// TIA Portal V19 export
FUNCTION "FC_EM_Plate" : Void   // FC4, FBD
{ S7_Optimized_Access := 'TRUE' }
// stored: SetENOAutomatically false
   VAR_TEMP
      Debug : Bool;
   END_VAR
BEGIN

REGION Network 1: ------------------------------------------------------------------------ Inputs ------------------------------------------------------------------------
END_REGION

REGION Network 2: Verwerken iPlateSenCilPushingIn_d0
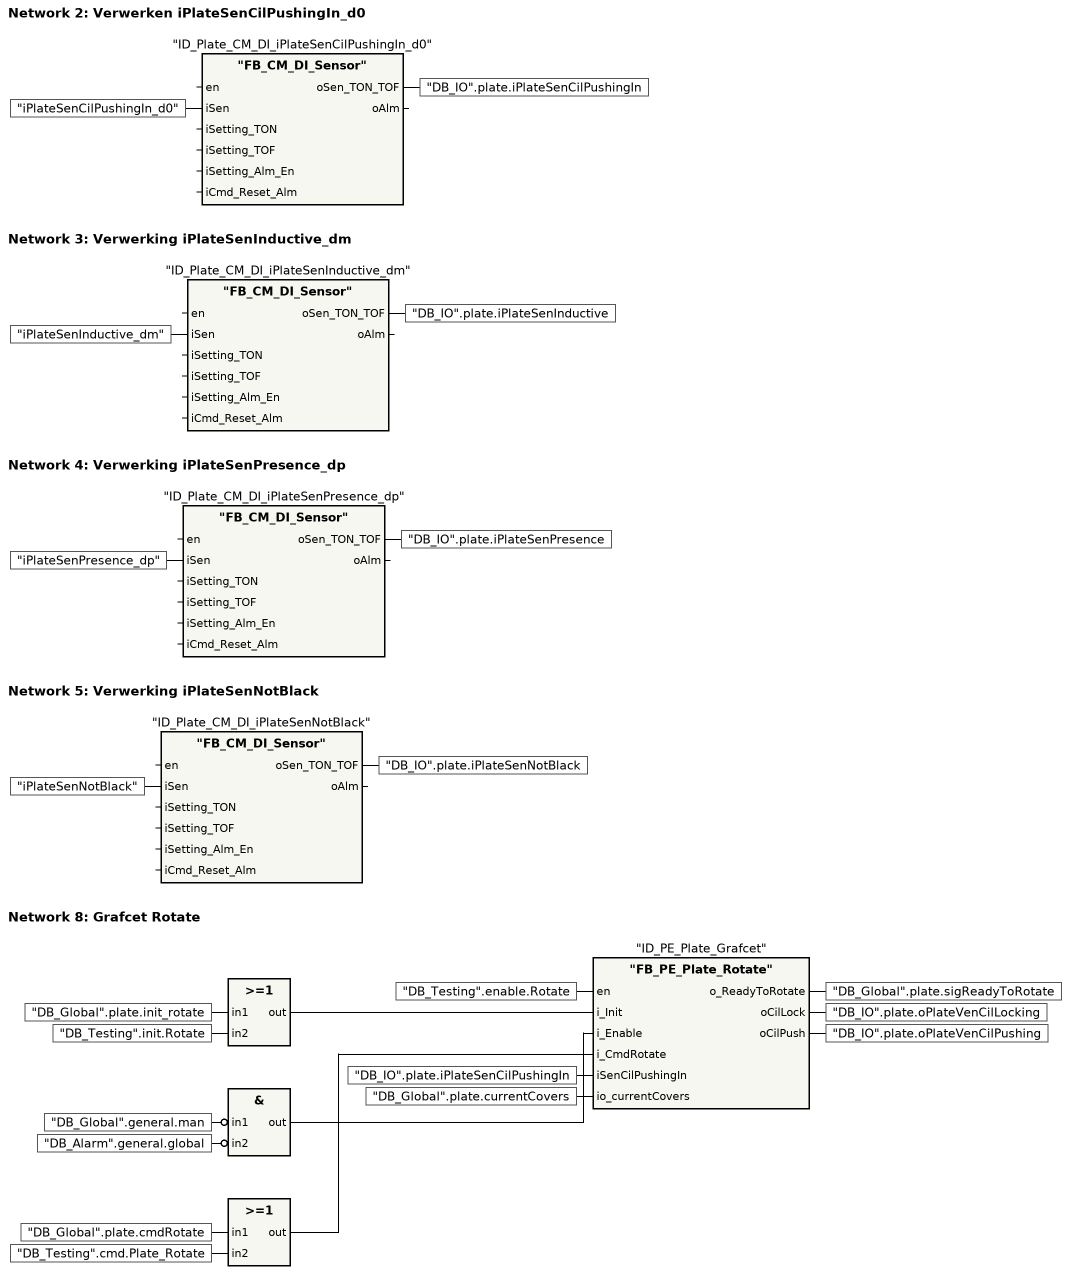
   "ID_Plate_CM_DI_iPlateSenCilPushingIn_d0"(iSen := "iPlateSenCilPushingIn_d0",   // "FB_CM_DI_Sensor"
                           oSen_TON_TOF => "DB_IO".plate.iPlateSenCilPushingIn);
END_REGION

REGION Network 3: Verwerking iPlateSenInductive_dm
   "ID_Plate_CM_DI_iPlateSenInductive_dm"(iSen := "iPlateSenInductive_dm",   // "FB_CM_DI_Sensor"
                           oSen_TON_TOF => "DB_IO".plate.iPlateSenInductive);
END_REGION

REGION Network 4: Verwerking iPlateSenPresence_dp
   "ID_Plate_CM_DI_iPlateSenPresence_dp"(iSen := "iPlateSenPresence_dp",   // "FB_CM_DI_Sensor"
                           oSen_TON_TOF => "DB_IO".plate.iPlateSenPresence);
END_REGION

REGION Network 5: Verwerking iPlateSenNotBlack
   "ID_Plate_CM_DI_iPlateSenNotBlack"(iSen := "iPlateSenNotBlack",   // "FB_CM_DI_Sensor"
                           oSen_TON_TOF => "DB_IO".plate.iPlateSenNotBlack);
END_REGION

REGION Network 6 (SCL): Verwerking iPlateSenHeight
   "DB_IO".plate.iPlateSenHeight := "iPlateSenHeight";
END_REGION

REGION Network 7: ------------------------------------------------------------------------ Logic ------------------------------------------------------------------------
END_REGION

REGION Network 8: Grafcet Rotate
   IF "DB_Testing".enable.Rotate THEN
       "ID_PE_Plate_Grafcet"(i_Init := "DB_Global".plate.init_rotate OR "DB_Testing".init.Rotate,   // "FB_PE_Plate_Rotate"
                             i_Enable := NOT "DB_Global".general.man AND NOT "DB_Alarm".general.global,
                             i_CmdRotate := "DB_Global".plate.cmdRotate OR "DB_Testing".cmd.Plate_Rotate,
                             iSenCilPushingIn := "DB_IO".plate.iPlateSenCilPushingIn,
                             io_currentCovers := "DB_Global".plate.currentCovers,
                             o_ReadyToRotate => "DB_Global".plate.sigReadyToRotate,
                             oCilLock => "DB_IO".plate.oPlateVenCilLocking,
                             oCilPush => "DB_IO".plate.oPlateVenCilPushing);
   END_IF;
END_REGION

REGION Network 9: Grafcet Measure
   // TODO:
   // - Correct placement in array
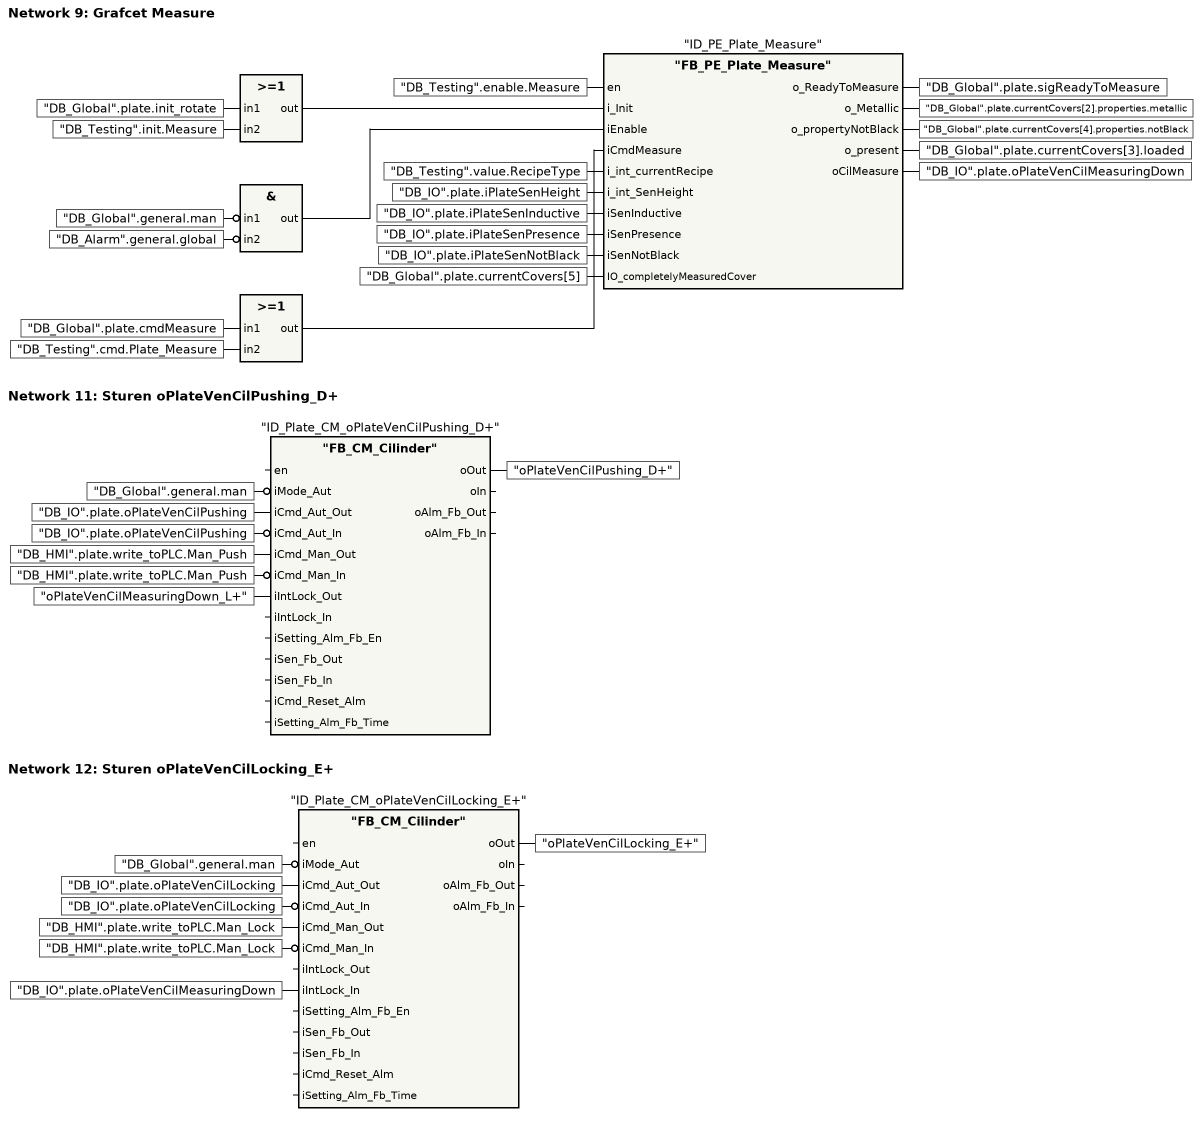
   IF "DB_Testing".enable.Measure THEN
       "ID_PE_Plate_Measure"(i_Init := "DB_Global".plate.init_rotate OR "DB_Testing".init.Measure,   // "FB_PE_Plate_Measure"
                             iEnable := NOT "DB_Global".general.man AND NOT "DB_Alarm".general.global,
                             iCmdMeasure := "DB_Global".plate.cmdMeasure OR "DB_Testing".cmd.Plate_Measure,
                             i_int_currentRecipe := "DB_Testing".value.RecipeType,
                             i_int_SenHeight := "DB_IO".plate.iPlateSenHeight,
                             iSenInductive := "DB_IO".plate.iPlateSenInductive,
                             iSenPresence := "DB_IO".plate.iPlateSenPresence,
                             iSenNotBlack := "DB_IO".plate.iPlateSenNotBlack,
                             IO_completelyMeasuredCover := "DB_Global".plate.currentCovers[5],
                             o_ReadyToMeasure => "DB_Global".plate.sigReadyToMeasure,
                             o_Metallic => "DB_Global".plate.currentCovers[2].properties.metallic,
                             o_propertyNotBlack => "DB_Global".plate.currentCovers[4].properties.notBlack,
                             o_present => "DB_Global".plate.currentCovers[3].loaded,
                             oCilMeasure => "DB_IO".plate.oPlateVenCilMeasuringDown);
   END_IF;
END_REGION

REGION Network 10: ------------------------------------------------------------------------ Outputs ------------------------------------------------------------------------
END_REGION

REGION Network 11: Sturen oPlateVenCilPushing_D+
   "ID_Plate_CM_oPlateVenCilPushing_D+"(iMode_Aut := NOT "DB_Global".general.man,   // "FB_CM_Cilinder"
                           iCmd_Aut_Out := "DB_IO".plate.oPlateVenCilPushing,
                           iCmd_Aut_In := NOT "DB_IO".plate.oPlateVenCilPushing,
                           iCmd_Man_Out := "DB_HMI".plate.write_toPLC.Man_Push,
                           iCmd_Man_In := NOT "DB_HMI".plate.write_toPLC.Man_Push,
                           iIntLock_Out := "oPlateVenCilMeasuringDown_L+",
                           oOut => "oPlateVenCilPushing_D+");
END_REGION

REGION Network 12: Sturen oPlateVenCilLocking_E+
   "ID_Plate_CM_oPlateVenCilLocking_E+"(iMode_Aut := NOT "DB_Global".general.man,   // "FB_CM_Cilinder"
                           iCmd_Aut_Out := "DB_IO".plate.oPlateVenCilLocking,
                           iCmd_Aut_In := NOT "DB_IO".plate.oPlateVenCilLocking,
                           iCmd_Man_Out := "DB_HMI".plate.write_toPLC.Man_Lock,
                           iCmd_Man_In := NOT "DB_HMI".plate.write_toPLC.Man_Lock,
                           iIntLock_In := "DB_IO".plate.oPlateVenCilMeasuringDown,
                           oOut => "oPlateVenCilLocking_E+");
END_REGION

REGION Network 13: Sturen oPlateVenCilMeasuringDown_L+
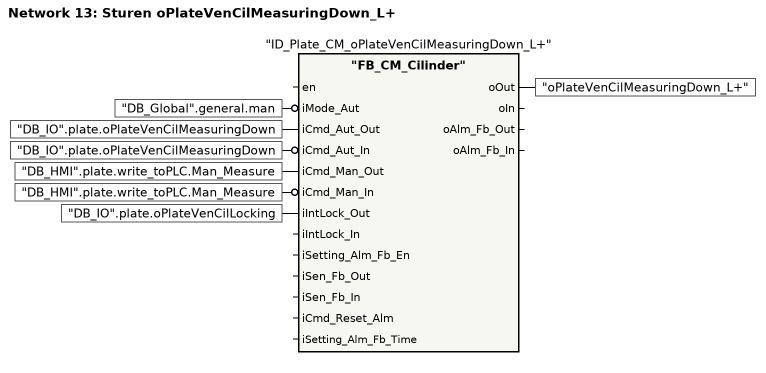
   "ID_Plate_CM_oPlateVenCilMeasuringDown_L+"(iMode_Aut := NOT "DB_Global".general.man,   // "FB_CM_Cilinder"
                           iCmd_Aut_Out := "DB_IO".plate.oPlateVenCilMeasuringDown,
                           iCmd_Aut_In := NOT "DB_IO".plate.oPlateVenCilMeasuringDown,
                           iCmd_Man_Out := "DB_HMI".plate.write_toPLC.Man_Measure,
                           iCmd_Man_In := NOT "DB_HMI".plate.write_toPLC.Man_Measure,
                           iIntLock_Out := "DB_IO".plate.oPlateVenCilLocking,
                           oOut => "oPlateVenCilMeasuringDown_L+");
END_REGION
END_FUNCTION
